ABB RobotStudio station: PracticaEntregable2EstacionDePartida.rsstn

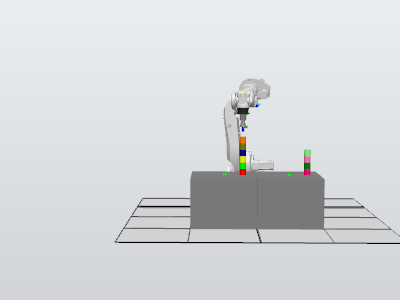
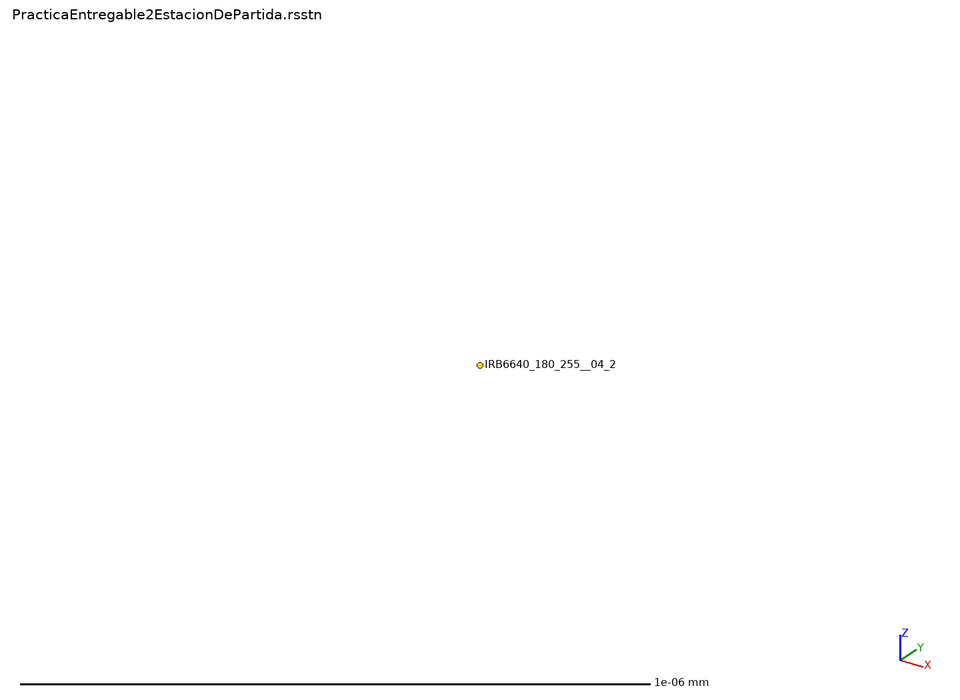
[picture v1: parts stored in the station drawn from their meshes, with robot base, taught points and paths (robot models come from the ABB library and are not in the file)]
Station Sesion3Prueba (saved by RobotStudio 24.1.10713.1)
Controller Controlador6
  mechanical unit ROB_1: IRB6640_180_255__04_2, 6 joints, base frame (0, 0, 0) mm
Layout (positions relative to the parent item):
  - Ventosa [mechanism] at (1500, -200, 1700) mm, rotated rx 180 ry 0 rz 180 deg
      TCP Ventosa at (0, 0, 200) mm
      links: PiezaVentosa
  - IRB6640_180_255__04_2 [mechanism, from %ABB.RobotStudio.Models.IRB6640%\IRB6640_180_255_G_04.rslib] at (0, 0, 0) mm; joint values [-0.1326, 0.0319, 0.1021, 0, 1.4368, -0.1326] (rad or m)
  - MesaTrabajoParteIzq [part], size 1000 x 1000 x 750 mm
  - MesaTrabajoParteDer [part], size 1000 x 1000 x 750 mm
  - Componente inteligente_1 [smart component]
      signals: DO Vacuostato, DI ActivaVentosa
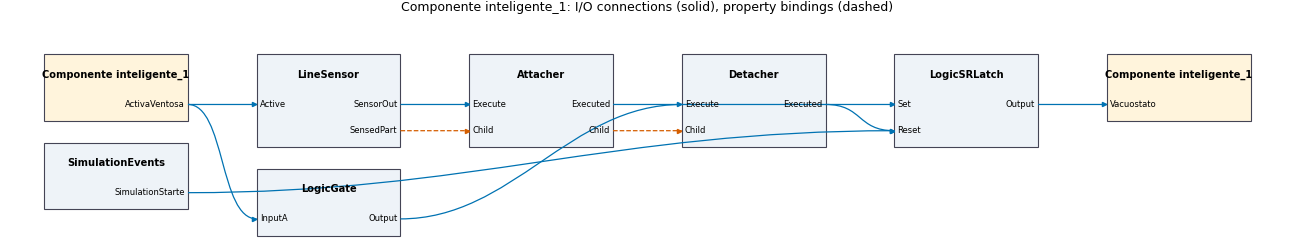
      connections:
        Componente inteligente_1.ActivaVentosa -> LineSensor.Active
        Componente inteligente_1.ActivaVentosa -> LogicGate.InputA
        LineSensor.SensorOut -> Attacher.Execute
        Attacher.Executed -> LogicSRLatch.Set
        LogicSRLatch.Output -> Componente inteligente_1.Vacuostato
        Detacher.Executed -> LogicSRLatch.Reset
        SimulationEvents.SimulationStarted -> LogicSRLatch.Reset
        LogicGate.Output -> Detacher.Execute
        LineSensor.SensedPart => Attacher.Child
        Attacher.Child => Detacher.Child
    - SimulationEvents [smart component, from Components\SimulationEvents.rslib]
    - LineSensor [smart component, from Components\LineSensor.rslib] at (1500, -200, 1500) mm, rotated rx 180 ry 0 rz 180 deg
        properties: Start=[0 0 -0.002]; End=[0 0 0.02]; Radius=0.002; SensedPart=Pieza_18; SensedPoint=[1.5 -0.200000030517578 1.35]; Length=0.022; Tag=(none)
      - _sensorPart_ [part], size 4 x 4 x 22 mm
    - LogicSRLatch [smart component, from Components\LogicSRLatch.rslib]
    - Attacher [smart component, from Components\Attacher.rslib]
        properties: Parent=Ventosa; Flange=0; Child=Pieza_18; Mount=false; Offset=[0 0 0]; Orientation=[0 0 0]
    - Detacher [smart component, from Components\Detacher.rslib]
        properties: Child=Pieza_18; KeepPosition=true
    - LogicGate [smart component, from Components\LogicGate.rslib]
        properties: Operator=NOT; Delay=0
  - Pieza_7 [part] at (0, 300, 0) mm, size 100 x 99.8 x 100 mm
  - Pieza_9 [part] at (0, 300, 100) mm, size 100 x 99.8 x 100 mm
  - Pieza_10 [part] at (0, 300, 200) mm, size 100 x 99.8 x 100 mm
  - Pieza_11 [part] at (0, 300, 300) mm, size 100 x 99.8 x 100 mm
  - Pieza_12 [part] at (0, 300, 0) mm, size 100 x 99.8 x 100 mm
  - Pieza_13 [part] at (0, 300, 100) mm, size 100 x 99.8 x 100 mm
  - Pieza_14 [part] at (0, 300, 200) mm, size 100 x 99.8 x 100 mm
  - Pieza_16 [part] at (0, 300, 300) mm, size 100 x 99.8 x 100 mm
  - Pieza_17 [part] at (0, 300, 400) mm, size 100 x 99.8 x 100 mm
  - Pieza_18 [part] at (0, 300, 500) mm, size 100 x 99.8 x 100 mm
Attachment: Ventosa is attached to IRB6640_180_255__04_2 / Link6
Attachment: LineSensor is attached to Ventosa / PiezaVentosa
Station logic (signal -> signal, property => property):
  Controlador6.SD_ActivaVentosa -> Componente inteligente_1.ActivaVentosa
  Componente inteligente_1.Vacuostato -> Controlador6.ED_PiezaCogida
Targets, tools, work objects and paths stored in the station, written as RAPID:
! task T_ROB1
MODULE CalibData
  PERS tooldata Ventosa:=[TRUE,[[0,0,200],[1,0,0,0]],[1,[0,0,125],[1,0,0,0],0,0,0.00125]];
ENDMODULE

! task T_ROB1
MODULE Module1
  CONST robtarget pBaseTorre1:=[[1500,500,750],[0,0,1,0],[0,0,0,0],[9E+09,9E+09,9E+09,9E+09,9E+09,9E+09]];
  CONST robtarget pBaseTorre2:=[[1500,-500,750],[0,0,1,0],[-1,0,-1,0],[9E+09,9E+09,9E+09,9E+09,9E+09,9E+09]];
  CONST robtarget pReposo:=[[1808.910161514,0,1855],[0.5,0,0.866025404,0],[0,0,0,0],[9E+09,9E+09,9E+09,9E+09,9E+09,9E+09]];
  PROC main()
    SetDO SD_ActivaVentosa,0;
    SetDO SD_ActivaVentosa,0;
  ENDPROC
ENDMODULE

